{attribute 'qualified_only'}
{attribute 'strict'}
TYPE E_EventType :
(
	None								:= 0,
	(* Normal StateMachine changes *)	
	SwitchOn 							:= 1,
	SwitchOff 							:= 2,
	HeatIsRequested 					:= 3,
	TargetTemperatureReached 			:= 4,
	CooledDown 							:= 5,
	Confirm 							:= 6,
	minWaterFlowReached					:= 7,
	
	(* Errors *)
	PressureDiffEvaporatorTooHigh		:= 101,
	EvaporatingTemperatureTooLow		:= 102,
	EvaporatingFlowRateTooLow			:= 103,
	LowPressureRefrigerationThermostat	:= 104,
	HighPressureRefrigerationThermostat	:= 105,
	MotorProtectionTriggered			:= 106,
	ExpansionValveTriggered				:= 107,
	IntermediateCircuitFlowRateTooLow	:= 108,
	LowPressureRefrigerationCalc		:= 109,
	TemperatureSourceWaterOutMinTooLow  := 110,
		
	(* Warnings *)
	HighPressureRefrigerationCalc		:= 202,
	WaterTankLevelTooLow				:= 203,
	WaterTankDataMissing				:= 204
);
END_TYPE

(* stored: Version 1.1.0.1
   DUT E_EventType: Id {7d29fffc-0140-4ddc-8b66-631419980f99} *)
